Yaskawa INFORM job: R1_W18,19,21(0,0)_KM-OK.JBI

/JOB
//NAME R1_W18,19,21(0,0)_KM-OK
///FOLDERNAME KRIS-SCIANA
//POS
///NPOS 130,130,0,7,0,0
///TOOL 0
///POSTYPE PULSE
///PULSE
C00000=114711,24992,37746,22148,54634,-40092
C00001=114711,25090,37980,22172,54546,-40112
C00002=116473,30887,46678,22230,51875,-39944
C00003=117693,37162,56822,22726,48755,-40141
C00004=117717,39214,58989,22811,48490,-40196
C00005=117162,33421,50450,22292,50747,-39900
C00006=124281,36200,51204,6663,52058,-33407
C00007=124281,37420,53845,6754,51066,-33474
C00008=123703,36737,50765,6834,52649,-33607
C00009=123224,33949,46516,6909,53863,-33722
C00010=121998,27604,36758,7127,56693,-34028
C00011=159186,30810,32621,13206,42177,-35854
C00012=160470,37862,42129,12809,39798,-35561
C00013=160967,40892,46239,12679,38772,-35459
C00014=161421,42558,49147,12571,37789,-35370
C00015=160967,40892,46239,12679,38772,-35459
C00016=154656,46922,57141,35742,37069,-45394
C00017=154381,49228,59680,36210,36875,-45681
C00018=154656,46922,57141,35742,37069,-45394
C00019=167044,45999,46410,-6240,44575,-27644
C00020=167633,46946,46573,-6596,45007,-27394
C00021=167044,45999,46410,-6240,44575,-27644
C00022=166770,42831,41934,-5939,45674,-27847
C00023=161065,21980,18252,-1988,49246,-30587
C00024=159647,45799,36518,69381,108582,-55306
C00025=158962,29647,19717,70315,101680,-54488
C00026=159831,31048,21110,70305,101039,-54439
C00027=160365,42547,32921,69473,106740,-56236
C00028=163700,38377,19102,57734,108457,-53162
C00029=164640,36884,17564,57835,107989,-52903
C00030=159571,51521,54149,76406,107689,-59893
C00031=162891,29266,7422,62096,107159,-52328
C00032=163286,27462,4647,62337,107291,-51925
C00033=162891,29266,7422,62096,107159,-52328
C00034=161898,29438,7023,62217,107944,-52356
C00035=157900,67762,47803,76590,91490,-60139
C00036=160086,65038,44626,76467,90101,-59697
C00037=160971,64038,43468,76405,89533,-59530
C00038=161808,65957,45694,76334,88844,-59627
C00039=160971,64038,43468,76405,89533,-59530
C00040=160746,61033,49335,86208,88631,-60628
C00041=161214,57780,45635,86203,88352,-60332
C00042=160746,61033,49335,86208,88631,-60628
C00043=159860,62185,50950,86211,89235,-60844
C00044=157670,65355,55356,86172,90720,-61418
C00045=149547,79598,79387,84947,95789,-65176
C00046=147380,29943,41067,-2068,90973,-56732
C00047=143824,33213,61180,-2695,80182,-57693
C00048=144583,34475,66777,-2587,77412,-57393
C00049=144894,35179,69272,-2544,76248,-57271
C00050=145794,38791,74922,-2403,74654,-56956
C00051=144894,35179,69272,-2544,76248,-57271
C00052=121537,9864,52031,32539,65160,-85705
C00053=121549,7365,49801,32520,65231,-85678
C00054=121151,9880,51545,32428,65555,-85731
C00055=120483,9209,49294,32124,66669,-85644
C00056=121381,7559,39748,31223,70673,-84112
C00057=124261,7577,20327,29903,80042,-80436
C00058=146234,20244,29766,39621,68335,-56412
C00059=157994,26355,46176,40344,57632,-55302
C00060=158938,27875,48706,40525,56611,-55292
C00061=159627,30276,52484,40896,55464,-55472
C00062=158938,27875,48706,40525,56611,-55292
C00063=161347,45131,60471,31596,68636,-55029
C00064=161865,42643,58570,31595,68356,-54903
C00065=161347,45131,60471,31596,68636,-55029
C00066=162067,35245,47673,33454,66786,-53625
C00067=163020,35202,46734,33229,66886,-53188
C00068=162067,35245,47673,33454,66786,-53625
C00069=161219,34196,45480,33361,67796,-53662
C00070=153721,32223,40712,33629,72334,-55377
C00071=124071,31447,57978,58015,40824,-35081
C00072=134905,36551,50551,5572,46905,-10907
C00073=134403,54808,77697,6663,39656,-11649
C00074=134154,54696,77991,6840,39438,-11789
C00075=125206,43446,60243,10751,45461,-15441
C00076=123261,39134,60266,12160,43538,-16593
C00077=130491,33558,34891,10462,68182,-18628
C00078=126810,29093,42144,49802,44475,-29714
C00079=134129,54590,77410,55610,35083,-32223
C00080=134174,53381,76001,55305,35202,-32051
C00081=133947,50704,72377,54403,35834,-31583
C00082=134636,54293,77964,56037,34514,-32383
C00083=132695,57663,83685,8012,37599,-12695
C00084=134144,54716,77911,6838,39499,-11786
C00085=130232,65613,97756,10545,33441,-14509
C00086=127586,39775,60949,9970,42882,-14628
C00087=124237,22307,34668,10410,50382,-15319
C00088=127823,12076,17182,44835,48527,-26383
C00089=139343,42729,17331,12753,96874,-21291
C00090=149144,58540,88158,21245,105799,-46112
C00091=153557,45831,57218,25770,116201,-42264
C00092=138732,36907,51372,33277,124468,-45980
C00093=139850,40077,70850,28601,111638,-49285
C00094=160392,54555,76642,27666,107314,-41703
C00095=160605,57503,80832,27595,106300,-41876
C00096=129561,32870,64605,21864,112431,-52912
C00097=129025,56334,93439,22167,113297,-53103
C00098=159827,52843,48366,24500,114532,-40726
C00099=157066,63408,96486,25008,101378,-44283
C00100=160961,54460,77288,27865,106738,-41632
C00101=153125,44530,54538,42337,119857,-40672
C00102=157404,15768,12223,35163,114278,-40456
C00103=160364,54759,76879,27645,107287,-41721
C00104=160577,57722,81090,27574,106268,-41895
C00105=141062,15534,36456,26515,108935,-49038
C00106=157776,59394,90985,21268,102261,-43972
C00107=160972,54368,77183,23536,106941,-41936
C00108=161021,60847,32788,71661,91289,-58028
C00109=158071,42272,26850,85179,79726,-64183
C00110=159982,40910,25376,84977,78370,-64008
C00111=160407,59632,31901,71739,91677,-58132
C00112=160676,63082,35844,71667,91272,-58387
C00113=160022,52515,61592,88250,76818,-71686
C00114=151897,58426,66630,87129,82620,-71919
C00115=158751,51722,59033,87847,77807,-71164
C00116=159892,50938,58162,87958,76997,-71072
C00117=160407,59632,31901,71739,91677,-58132
C00118=160676,63082,35844,71667,91272,-58387
C00119=160063,48160,52262,87506,77036,-70029
C00120=151932,45808,25021,85459,84488,-63059
C00121=157434,41112,20051,84712,80618,-62540
C00122=160036,40278,19462,84376,78747,-62460
C00123=160407,59632,31901,71739,91677,-58132
C00124=160676,63082,35844,71667,91272,-58387
C00125=160053,50810,58014,87970,76885,-71060
C00126=156942,58566,66790,87841,79014,-71800
C00127=144428,79961,92656,86096,87446,-74437
C00128=71141,-66575,-39760,86096,87446,-74437
C00129=10106,-66575,-39760,6607,87446,-74437
BC00000=310143,434635,881827
BC00001=310143,415745,591140
BC00002=310143,415745,591140
BC00003=310143,415746,591137
BC00004=310143,415746,591137
BC00005=310143,415745,591140
BC00006=310143,415745,591140
BC00007=310143,415745,591140
BC00008=310143,415745,591140
BC00009=310143,415745,591140
BC00010=310143,415745,591140
BC00011=311385,408712,898001
BC00012=311385,408712,898001
BC00013=311385,408712,898001
BC00014=311385,408712,898001
BC00015=311385,408712,898001
BC00016=311385,408712,898001
BC00017=311385,408712,898001
BC00018=311385,408712,898001
BC00019=311385,408712,898001
BC00020=311385,408712,898001
BC00021=311385,408712,898001
BC00022=311385,408712,898001
BC00023=311385,408712,898001
BC00024=327465,406418,676623
BC00025=327465,406418,676623
BC00026=327465,406418,676623
BC00027=327465,406418,676623
BC00028=327465,406418,676623
BC00029=327465,406418,676623
BC00030=327465,406418,676623
BC00031=327465,406418,676623
BC00032=327465,406418,676623
BC00033=327465,406418,676623
BC00034=327465,406418,676623
BC00035=365912,447627,1041849
BC00036=365912,447627,1041849
BC00037=365912,447627,1041849
BC00038=365912,447627,1041849
BC00039=365912,447627,1041849
BC00040=365912,447627,1041849
BC00041=365912,447627,1041849
BC00042=365912,447627,1041849
BC00043=365912,447627,1041849
BC00044=365912,447627,1041849
BC00045=365912,447627,1041849
BC00046=325049,437381,764783
BC00047=325049,437381,764783
BC00048=325049,437381,764783
BC00049=325049,437381,764783
BC00050=325049,437381,764783
BC00051=325049,437381,764783
BC00052=325049,437381,764783
BC00053=325049,437381,764783
BC00054=325049,437381,764783
BC00055=325049,437381,764783
BC00056=325049,437381,764783
BC00057=325049,437381,764783
BC00058=319824,453964,991370
BC00059=319824,453964,991370
BC00060=319824,453964,991370
BC00061=319824,453964,991370
BC00062=319824,453964,991370
BC00063=319824,453964,991370
BC00064=319824,453964,991370
BC00065=319824,453964,991370
BC00066=319824,453964,991370
BC00067=319824,453964,991370
BC00068=319824,453964,991370
BC00069=319824,453964,991370
BC00070=319824,453964,991370
BC00071=249698,446219,1049528
BC00072=245232,432157,891860
BC00073=245232,432157,891860
BC00074=270365,431987,815579
BC00075=270365,431987,707001
BC00076=271418,434166,822270
BC00077=289749,434611,781176
BC00078=249740,446224,941994
BC00079=244219,441045,935155
BC00080=242011,438973,932420
BC00081=242011,438973,932420
BC00082=242011,438973,932420
BC00083=196339,432488,1040261
BC00084=232937,432240,929179
BC00085=232936,432241,929176
BC00086=233991,434420,935870
BC00087=236625,439870,952599
BC00088=286889,445967,936649
BC00089=311361,435135,732726
BC00090=306652,384495,984795
BC00091=306653,384495,802379
BC00092=269816,393303,755996
BC00093=269816,393304,824894
BC00094=302387,393083,859863
BC00095=302387,393083,859863
BC00096=285064,393304,712701
BC00097=285064,393304,712701
BC00098=331782,386257,791590
BC00099=274081,384716,1075175
BC00100=274122,384721,976120
BC00101=269816,393304,824894
BC00102=269816,393304,824894
BC00103=269816,393304,958722
BC00104=269816,393304,958722
BC00105=269816,393304,824894
BC00106=299213,386462,890339
BC00107=299172,386457,997874
BC00108=368384,441548,1075175
BC00109=360608,449199,1075175
BC00110=360608,449199,1075175
BC00111=360608,449199,1075175
BC00112=360608,449199,1075175
BC00113=360608,449199,1075175
BC00114=360608,449199,871920
BC00115=360608,449199,871920
BC00116=360608,449199,871920
BC00117=360608,449199,1075175
BC00118=360608,449199,1075175
BC00119=360608,449199,655426
BC00120=360609,449199,890554
BC00121=360609,449199,890554
BC00122=360608,449199,890556
BC00123=360608,449199,1075175
BC00124=360608,449199,1075175
BC00125=360608,449199,871921
BC00126=360608,449199,871921
BC00127=360608,449199,871921
BC00128=360608,449199,871921
BC00129=221411,449199,1015609
///POSTYPE BASE
///RECTAN
///RCONF 0,0,0,0,1,0,0,0,0,0,0,0,0,0,0,0,0,0,0,0,0,0,0,0
P00006=2.006,1.622,-0.565,0.0000,0.0000,0.0000
P00021=0.073,2.058,-0.109,0.0000,0.0000,0.0000
P00022=2.006,1.622,-0.565,0.0000,0.0000,0.0000
///RCONF 0,0,0,0,0,0,0,0,0,0,0,0,0,0,0,0,0,0,0,0,0,0,0,0
P00023=-2.957,-4.083,2.762,0.0000,0.0000,0.0000
P00024=-1.466,-0.226,-0.419,0.0000,0.0000,0.0000
P00025=3.643,0.007,-2.585,0.0000,0.0000,0.0000
P00026=2.644,0.055,-2.583,0.0000,0.0000,0.0000
//INST
///DATE 2023/12/14 11:02
///ATTR SC,RW
///GROUP1 RB1,BS1
NOP
SFTOF
MOVJ C00000 BC00000 VJ=100.00
MOVJ C00001 BC00001 VJ=100.00
MOVJ C00002 BC00002 VJ=100.00
MOVL C00003 BC00003 V=60.0
REFP 3 C00004 BC00004
CALL JOB:SEARCH-R1
SET P021 P006
SFTON P021
MOVL C00005 BC00005 V=60.0
MOVL C00006 BC00006 V=60.0
REFP 3 C00007 BC00007
CALL JOB:SEARCH-R1
SET P021 P006
SFTON P021
MOVL C00008 BC00008 V=60.0
MOVL C00009 BC00009 V=100.0
MOVL C00010 BC00010 V=100.0
'Path S876 (for W416)
SFTOF
MOVL C00011 BC00011 V=333.3
MOVJ C00012 BC00012 VJ=100.00
MOVL C00013 BC00013 V=60.0
REFP 3 C00014 BC00014
CALL JOB:SEARCH-R1
SET P022 P006
SFTON P022
MOVL C00015 BC00015 V=60.0
MOVL C00016 BC00016 V=60.0
REFP 3 C00017 BC00017
CALL JOB:SEARCH-R1
SET P022 P006
SFTON P022
MOVL C00018 BC00018 V=60.0
MOVL C00019 BC00019 V=60.0
REFP 3 C00020 BC00020
CALL JOB:SEARCH-R1
SET P022 P006
SFTON P022
MOVL C00021 BC00021 V=60.0
MOVL C00022 BC00022 V=100.0
MOVL C00023 BC00023 V=100.0
'Path S877 (for W886)
SFTOF
MOVL C00024 BC00024 V=250.0
MOVL C00025 BC00025 V=83.3
REFP 3 C00026 BC00026
CALL JOB:SEARCH-R1
SET P025 P006
SFTON P025
MOVL C00027 BC00027 V=60.0
MOVL C00028 BC00028 V=60.0
REFP 3 C00029 BC00029
CALL JOB:SEARCH-R1
SET P025 P006
SFTON P025
MOVL C00030 BC00030 V=60.0
MOVL C00031 BC00031 V=60.0
REFP 3 C00032 BC00032
CALL JOB:SEARCH-R1
SET P025 P006
SFTON P025
MOVL C00033 BC00033 V=60.0
MOVL C00034 BC00034 V=100.0
'Path S878 (for W886)
SFTOF
MOVL C00035 BC00035 V=333.3
MOVL C00036 BC00036 V=166.7
MOVL C00037 BC00037 V=60.0
REFP 3 C00038 BC00038
CALL JOB:SEARCH-R1
SET P026 P006
SFTON P026
MOVL C00039 BC00039 V=60.0
MOVL C00040 BC00040 V=60.0
REFP 3 C00041 BC00041
CALL JOB:SEARCH-R1
SET P026 P006
SFTON P026
MOVL C00042 BC00042 V=60.0
MOVL C00043 BC00043 V=100.0
MOVL C00044 BC00044 V=166.7
'Path S879 (for W18)
SFTOF
MOVJ C00045 BC00045 VJ=100.00
MOVJ C00046 BC00046 VJ=100.00
MOVJ C00047 BC00047 VJ=100.00
MOVJ C00048 BC00048 VJ=100.00
MOVL C00049 BC00049 V=133.3
REFP 3 C00050 BC00050
CALL JOB:SEARCH-R1
SET P023 P006
SFTON P023
MOVL C00051 BC00051 V=60.0
MOVL C00052 BC00052 V=100.0
REFP 3 C00053 BC00053
CALL JOB:SEARCH-R1
SET P023 P006
SFTON P023
MOVL C00054 BC00054 V=60.0
MOVL C00055 BC00055 V=100.0
MOVL C00056 BC00056 V=250.0
'Path S880 (for W18)
SFTOF
MOVJ C00057 BC00057 VJ=100.00
MOVJ C00058 BC00058 VJ=100.00
MOVJ C00059 BC00059 VJ=100.00
MOVL C00060 BC00060 V=60.0
REFP 3 C00061 BC00061
CALL JOB:SEARCH-R1
SET P024 P006
SFTON P024
MOVL C00062 BC00062 V=60.0
MOVL C00063 BC00063 V=60.0
REFP 3 C00064 BC00064
CALL JOB:SEARCH-R1
SET P024 P006
SFTON P024
MOVL C00065 BC00065 V=60.0
MOVL C00066 BC00066 V=60.0
REFP 3 C00067 BC00067
CALL JOB:SEARCH-R1
SET P024 P006
SFTON P024
MOVL C00068 BC00068 V=60.0
MOVL C00069 BC00069 V=100.0
MOVL C00070 BC00070 V=250.0
'Path W881
SFTOF
MOVJ C00071 BC00071 VJ=100.00
MOVL C00072 BC00072 V=166.7
MOVL C00073 BC00073 V=166.7
MACRO1 MJ#(0) ARGF10
ARCON
MOVL C00074 BC00074 V=13.3
MOVL C00075 BC00075 V=13.3
ARCOF
MOVL C00076 BC00076 V=166.7
MOVJ C00077 BC00077 VJ=100.00
SFTOF
SFTON P021
MOVJ C00078 BC00078 VJ=100.00
MOVL C00079 BC00079 V=250.0
MOVL C00080 BC00080 V=100.0 PL=0
REFP 1 C00081 BC00081
REFP 2 C00082 BC00082
MACRO1 MJ#(0) ARGF10
ARCON
MOVL C00083 BC00083 V=13.3
MOVL C00084 BC00084 V=13.3
MOVL C00085 BC00085 V=13.3
ARCOF
MOVL C00086 BC00086 V=166.7
MOVL C00087 BC00087 V=250.0
SFTOF
'Path W921
SFTOF
MOVJ C00088 BC00088 VJ=100.00
SFTON P021
'Path VIA889
SFTOF
MOVJ C00089 BC00089 VJ=100.00
'Path W922_19A
SFTOF
SFTON P024
MOVJ C00090 BC00090 VJ=100.00
MOVJ C00091 BC00091 VJ=100.00
MOVL C00092 BC00092 V=100.0
MOVL C00093 BC00093 V=100.0 PL=0
REFP 1 C00094 BC00094
REFP 2 C00095 BC00095
MACRO1 MJ#(0) ARGF10
ARCON
MOVL C00096 BC00096 V=13.3
ARCOF
MOVL C00097 BC00097 V=100.0
MOVL C00098 BC00098 V=250.0
SFTOF
'Path W882_19B
SFTOF
SFTON P024
MOVJ C00099 BC00099 VJ=100.00
MOVJ C00100 BC00100 VJ=100.00
MOVL C00101 BC00101 V=250.0
MOVL C00102 BC00102 V=100.0 PL=0
REFP 1 C00103 BC00103
REFP 2 C00104 BC00104
MACRO1 MJ#(0) ARGF10
ARCON
MOVL C00105 BC00105 V=13.3
ARCOF
MOVL C00106 BC00106 V=100.0
MOVL C00107 BC00107 V=333.3
SFTOF
'Path W883_A
SFTOF
SFTON P026
MOVL C00108 BC00108 V=333.3
MOVL C00109 BC00109 V=250.0
MOVL C00110 BC00110 V=166.7 PL=0
REFP 1 C00111 BC00111
REFP 2 C00112 BC00112
MACRO1 MJ#(0) ARGF6
ARCON
MOVL C00113 BC00113 V=13.3
ARCOF
'Path W883_C
SFTOF
SFTON P026
MOVL C00114 BC00114 V=100.0
MOVL C00115 BC00115 V=100.0
MOVL C00116 BC00116 V=100.0 PL=0
REFP 1 C00117 BC00117
REFP 2 C00118 BC00118
MACRO1 MJ#(0) ARGF6
ARCON
MOVL C00119 BC00119 V=13.3
ARCOF
'Path W883_B
SFTOF
SFTON P026
MOVL C00120 BC00120 V=100.0
MOVL C00121 BC00121 V=100.0
MOVL C00122 BC00122 V=100.0 PL=0
REFP 1 C00123 BC00123
REFP 2 C00124 BC00124
MACRO1 MJ#(0) ARGF6
ARCON
MOVL C00125 BC00125 V=13.3
ARCOF
MOVL C00126 BC00126 V=100.0
SFTOF
MOVL C00127 BC00127 V=100.0
MOVJ C00128 BC00128 VJ=100.00
MOVJ C00129 BC00129 VJ=100.00
END
